% RSLogix 500 project Servo Control for Automated Valve Sequencing.RSS, saved by version 8.30.00.16 %
PROJECT "UNTITLED"    % processor: Bul.1763 MicroLogix 1100 Series B %

PROGRAM FILES
  LAD 2 "MAIN"  3 rungs
  LAD 3 "IO"  7 rungs
  LAD 4 "CTRLS"  12 rungs

DATA FILES
  O0 OUTPUT  4 elements
  I1 INPUT  6 elements
  S2 STATUS  66 elements
  B3 BINARY  2 elements
  T4 TIMER  3 elements
  C5 COUNTER  1 elements
  R6 CONTROL  1 elements
  N7 INTEGER  1 elements
  F8 FLOAT  1 elements

LADDER 2 "MAIN"
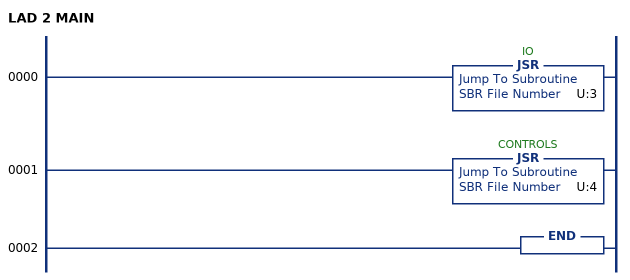
% Rung: 0 %
SOR JSR U:3 EOR
%   U:3  "IO" %
% Rung: 1 %
SOR JSR U:4 EOR
%   U:4  "CONTROLS" %
% Rung: 2 %
SOR END EOR

LADDER 3 "IO"
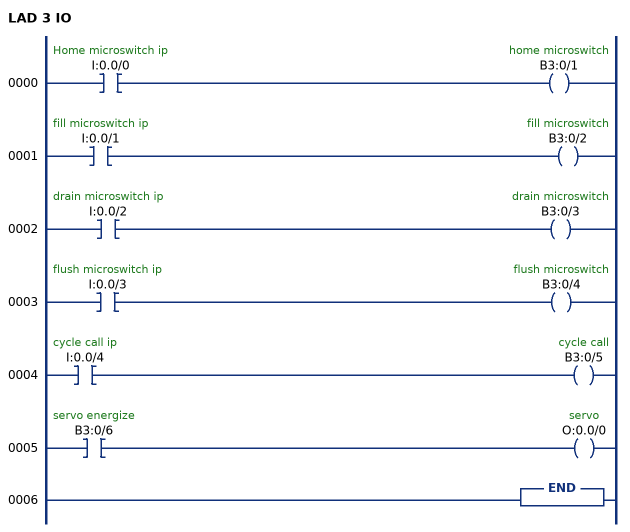
% Rung: 0 %
SOR XIC I:0.0/0 OTE B3:0/1 EOR
%   I:0.0/0  "Home microswitch ip" %
%   B3:0/1  "home microswitch" %
% Rung: 1 %
SOR XIC I:0.0/1 OTE B3:0/2 EOR
%   I:0.0/1  "fill microswitch ip" %
%   B3:0/2  "fill microswitch" %
% Rung: 2 %
SOR XIC I:0.0/2 OTE B3:0/3 EOR
%   I:0.0/2  "drain microswitch ip" %
%   B3:0/3  "drain microswitch" %
% Rung: 3 %
SOR XIC I:0.0/3 OTE B3:0/4 EOR
%   I:0.0/3  "flush microswitch ip" %
%   B3:0/4  "flush microswitch" %
% Rung: 4 %
SOR XIC I:0.0/4 OTE B3:0/5 EOR
%   I:0.0/4  "cycle call ip" %
%   B3:0/5  "cycle call" %
% Rung: 5 %
SOR XIC B3:0/6 OTE O:0.0/0 EOR
%   B3:0/6  "servo energize" %
%   O:0.0/0  "servo" %
% Rung: 6 %
SOR END EOR

LADDER 4 "CTRLS"
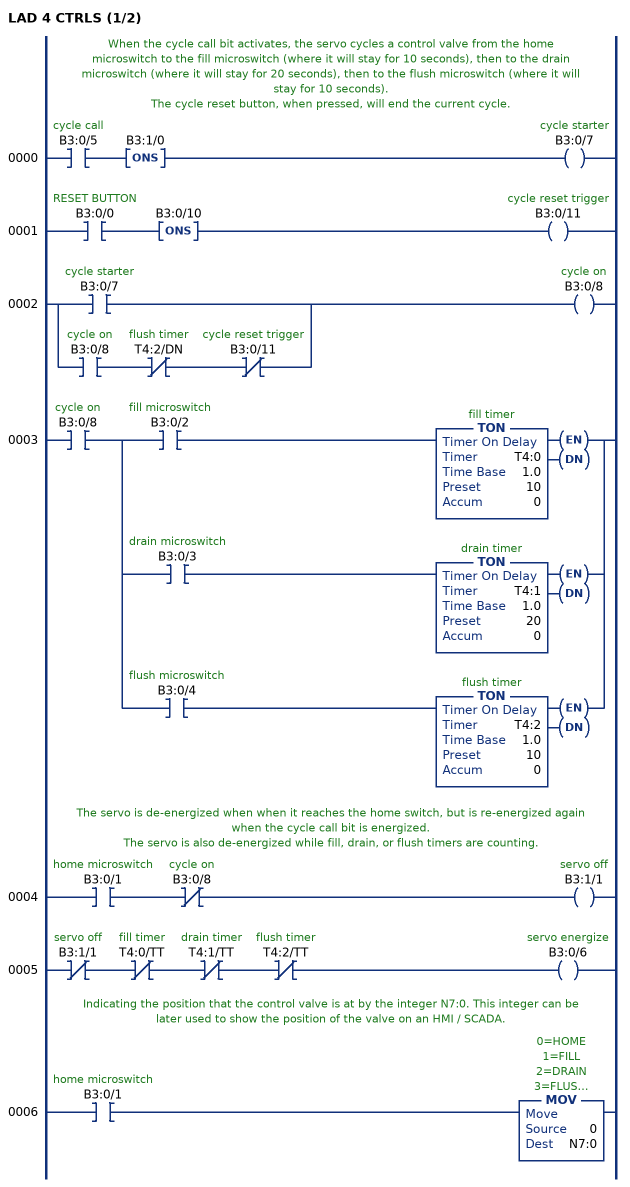
% Rung: 0 %
% When the cycle call bit activates, the servo cycles a control valve from the home microswitch to the fill microswitch (where it will stay for 10 seconds), then to the drain microswitch (where it will stay for 20 seconds), then to the flush microswitch (where it will stay for 10 seconds).
% The cycle reset button, when pressed, will end the current cycle. %
SOR XIC B3:0/5 ONS B3:1/0 OTE B3:0/7 EOR
%   B3:0/5  "cycle call" %
%   B3:0/7  "cycle starter" %
% Rung: 1 %
SOR XIC B3:0/0 ONS B3:0/10 OTE B3:0/11 EOR
%   B3:0/0  "RESET BUTTON" %
%   B3:0/11  "cycle reset trigger" %
% Rung: 2 %
SOR BST XIC B3:0/7 NXB XIC B3:0/8 XIO T4:2/DN XIO B3:0/11 BND OTE B3:0/8 EOR
%   B3:0/7  "cycle starter" %
%   B3:0/8  "cycle on" %
%   T4:2  "flush timer" %
%   B3:0/11  "cycle reset trigger" %
% Rung: 3 %
SOR XIC B3:0/8 BST XIC B3:0/2 TON T4:0 1.0 10 0 NXB XIC B3:0/3 TON T4:1 1.0 20 0 NXB XIC B3:0/4 TON T4:2 1.0 10 0 BND EOR
%   B3:0/8  "cycle on" %
%   B3:0/2  "fill microswitch" %
%   T4:0  "fill timer" %
%   B3:0/3  "drain microswitch" %
%   T4:1  "drain timer" %
%   B3:0/4  "flush microswitch" %
%   T4:2  "flush timer" %
% Rung: 4 %
% The servo is de-energized when when it reaches the home switch, but is re-energized again when the cycle call bit is energized.
% The servo is also de-energized while fill, drain, or flush timers are counting. %
SOR XIC B3:0/1 XIO B3:0/8 OTE B3:1/1 EOR
%   B3:0/1  "home microswitch" %
%   B3:0/8  "cycle on" %
%   B3:1/1  "servo off" %
% Rung: 5 %
SOR XIO B3:1/1 XIO T4:0/TT XIO T4:1/TT XIO T4:2/TT OTE B3:0/6 EOR
%   B3:1/1  "servo off" %
%   T4:0  "fill timer" %
%   T4:1  "drain timer" %
%   T4:2  "flush timer" %
%   B3:0/6  "servo energize" %
% Rung: 6 %
% Indicating the position that the control valve is at by the integer N7:0. This integer can be later used to show the position of the valve on an HMI / SCADA. %
SOR XIC B3:0/1 MOV 0 N7:0 EOR
%   B3:0/1  "home microswitch" %
%   N7:0  "0=HOME 1=FILL 2=DRAIN 3=FLUSH 4=TRAVELLING" %

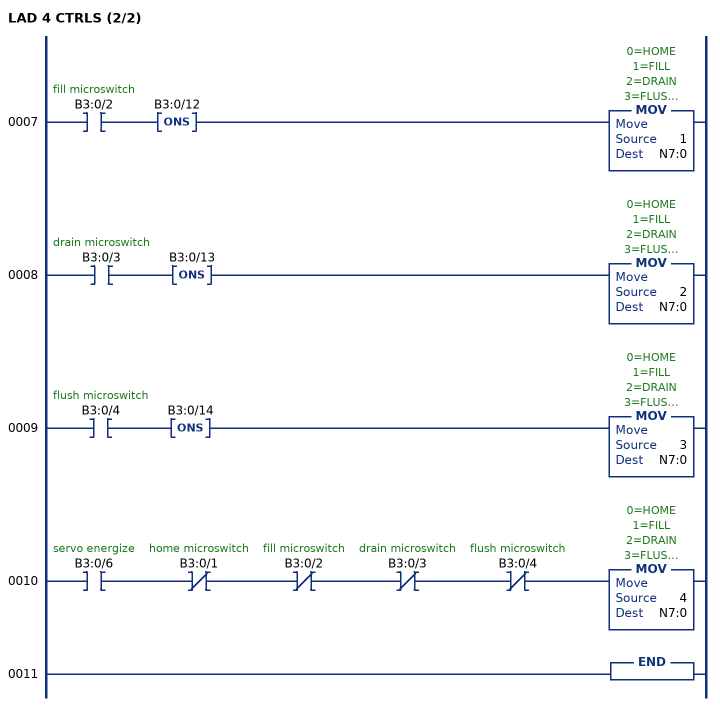
% Rung: 7 %
SOR XIC B3:0/2 ONS B3:0/12 MOV 1 N7:0 EOR
%   B3:0/2  "fill microswitch" %
%   N7:0  "0=HOME 1=FILL 2=DRAIN 3=FLUSH 4=TRAVELLING" %
% Rung: 8 %
SOR XIC B3:0/3 ONS B3:0/13 MOV 2 N7:0 EOR
%   B3:0/3  "drain microswitch" %
%   N7:0  "0=HOME 1=FILL 2=DRAIN 3=FLUSH 4=TRAVELLING" %
% Rung: 9 %
SOR XIC B3:0/4 ONS B3:0/14 MOV 3 N7:0 EOR
%   B3:0/4  "flush microswitch" %
%   N7:0  "0=HOME 1=FILL 2=DRAIN 3=FLUSH 4=TRAVELLING" %
% Rung: 10 %
SOR XIC B3:0/6 XIO B3:0/1 XIO B3:0/2 XIO B3:0/3 XIO B3:0/4 MOV 4 N7:0 EOR
%   B3:0/6  "servo energize" %
%   B3:0/1  "home microswitch" %
%   B3:0/2  "fill microswitch" %
%   B3:0/3  "drain microswitch" %
%   B3:0/4  "flush microswitch" %
%   N7:0  "0=HOME 1=FILL 2=DRAIN 3=FLUSH 4=TRAVELLING" %
% Rung: 11 %
SOR END EOR

DATA TABLE (non-zero values as saved)
DATA T4
% .PRE .ACC %
% T4:0 % 10 0
% T4:1 % 20 0
% T4:2 % 10 0
